// TIA Portal V20 export
TYPE "LKinCtrl_Utilities_typeSearchableTableConfiguration"
// stored: Access Published
   STRUCT
      numberOfElements { ExternalAccessible := 'False'; ExternalVisible := 'False'; ExternalWritable := 'False'} : DInt := -1;   // Total number of elements to be considered. If smaller or bigger than searchMask maximum is taken.
      emptyTable { ExternalAccessible := 'False'; ExternalVisible := 'False'; ExternalWritable := 'False'} : Bool;   // TRUE: The table is empty. No selection, no interactivity.
      sizeTableWindow { ExternalAccessible := 'False'; ExternalVisible := 'False'; ExternalWritable := 'False'} : USInt := 1;   // Number of elements that can be displayed at once in the table window.
      fieldsToSkip { ExternalAccessible := 'False'; ExternalVisible := 'False'; ExternalWritable := 'False'} : USInt := 1;   // Number of fields to skip when button up or down is pressed.
   END_STRUCT;
END_TYPE
